FUNCTION_BLOCK FB_TopElement_HMI EXTENDS FB_BaseTopElement_HMI IMPLEMENTS ITF_TopElement_HMI
VAR
	itfTopElementConnector				: ITF_TopElement_HMI_Connector;
	refstTopElementData					: REFERENCE TO ST_TopElement_HMI;
	itfControlElement1					: ITF_ControlElement_HMI;
	itfControlElement2					: ITF_ControlElement_HMI;
	itfGroupElement1					: ITF_GroupElement_HMI;
	itfComponent1						: ITF_Component_HMI;
	itfComponent2						: ITF_Component_HMI;
	itfComponent3						: ITF_Component_HMI;
END_VAR

METHOD FB_init : BOOL
VAR_INPUT
	bInitRetains : BOOL; // if TRUE, the retain variables are initialized (warm start / cold start)
	bInCopyCode : BOOL;  // if TRUE, the instance afterwards gets moved into the copy code (online change)
	itfBaseLoggerConnector				: ITF_BaseLogger_HMI_Connector;	//bezpośredni łącznik do logera
	itfTopElementConnector				: ITF_TopElement_HMI_Init;
	itfControlElement1					: ITF_ControlElement_HMI;
	itfControlElement2					: ITF_ControlElement_HMI;
	itfGroupElement1					: ITF_GroupElement_HMI;
	itfComponent1						: ITF_Component_HMI;
	itfComponent2						: ITF_Component_HMI;
	itfComponent3						: ITF_Component_HMI;
END_VAR
//Przypisanie do elementu który własnie stworzyliśmy
THIS^.itfTopElementConnector			:= itfTopElementConnector;
//Przypisanie do elementów z biblioteki
THIS^.itfBaseLoggerElementConnector		:= itfTopElementConnector;
THIS^.itfBaseComponentConnector			:= itfTopElementConnector;
THIS^.itfBaseControlElementConnector	:= itfTopElementConnector;
THIS^.itfBaseGroupElementConnector		:= itfTopElementConnector;
THIS^.itfBaseTopElementConnector		:= itfTopElementConnector;
//
THIS^.itfBaseLoggerConnector			:= itfBaseLoggerConnector;

THIS^.itfControlElement1				:= itfControlElement1;
THIS^.AddControlElement (itfControlElementHMI	:= itfControlElement1);
THIS^.itfControlElement2				:= itfControlElement2;
THIS^.AddControlElement (itfControlElementHMI	:= itfControlElement2);
THIS^.itfGroupElement1					:= itfGroupElement1;
THIS^.AddControlElement (itfControlElementHMI	:= itfGroupElement1);
THIS^.itfComponent1						:= itfComponent1;
THIS^.AddComponent (itfComponentHMI		:= itfComponent1);
THIS^.itfComponent2						:= itfComponent2;
THIS^.AddComponent (itfComponentHMI		:= itfComponent2);
THIS^.itfComponent3						:= itfComponent3;
THIS^.AddComponent (itfComponentHMI		:= itfComponent3);


IF (THIS^.itfTopElementConnector <> 0 AND
	THIS^.itfBaseLoggerElementConnector <> 0 AND
	THIS^.itfBaseComponentConnector	<> 0 AND
	THIS^.itfBaseControlElementConnector <> 0 AND
	THIS^.itfBaseGroupElementConnector <> 0 AND
	THIS^.itfBaseTopElementConnector <> 0 AND
	THIS^.itfBaseLoggerConnector <> 0) THEN
	THIS^.bIsInit						:= TRUE;
END_IF
END_METHOD

METHOD LinkTopElementData : BOOL
VAR_INPUT
	stData				: REFERENCE TO ST_TopElement_HMI_Link;
END_VAR
THIS^.refstTopElementData	REF= stData.stTopElement;

THIS^.refstBaseLoggerElementDataHMI	REF= stData.stBaseLoggerElement;
THIS^.refstBaseComponentDataHMI		REF= stData.stBaseComponent;
THIS^.refstBaseControlElementDataHMI	REF= stData.stBaseControlElement;
THIS^.refstBaseGroupElementDataHMI		REF= stData.stBaseGroupElement;
THIS^.refstBaseTopElementDataHMI		REF= stData.stBaseTopElement;

THIS^.itfControlElement1.LinkControlElementData (stData := stData.stControlElement1);
THIS^.itfControlElement2.LinkControlElementData (stData := stData.stControlElement2);
THIS^.itfGroupElement1.LinkGroupelementData (stData := stData.stGroupElement1);
THIS^.itfComponent1.LinkComponentData (stData := stData.stComponent1);
THIS^.itfComponent2.LinkComponentData (stData := stData.stComponent2);
THIS^.itfComponent3.LinkComponentData (stData := stData.stComponent3);

THIS^.CreateLinkToEventsMemory ();



IF (__ISVALIDREF (THIS^.refstTopElementData) AND this^.IsLinkedReferences ()) THEN
	THIS^.bIsValidData		:= TRUE;
	LinkTopElementData		:= TRUE;
END_IF
END_METHOD

END_FUNCTION_BLOCK

(* stored: Version 1.1.0.1, ProductVersion 3.1.4024.15
   POU FB_TopElement_HMI: Id {54abd47c-3eb0-49fb-a4d6-79dd6427523e}, SpecialFunc None
   Folder ITF_TopElement_HMI: Id {cc456a88-f147-42c3-b563-9e014e00639c}
   Method FB_init: Id {ee1e6a46-fdbb-4ec7-8f35-1725de8de569}
   Method LinkTopElementData: Id {b5b619bd-8b68-4908-b96b-4f1ab05bb941} *)
